FUNCTION WRITE_ANY_STRING : BOOL
VAR_INPUT
    ptr: POINTER TO STRING;
    val: STRING;
END_VAR

ptr^ := val;

END_FUNCTION

(* stored: Version 1.1.0.1, ProductVersion 3.1.4022.9
   POU WRITE_ANY_STRING: Id {bad90aed-e2f4-4920-ad52-32ebaec9fc44}, SpecialFunc None *)
